{attribute 'linkalways'} 
{attribute 'no_explicit_call' := 'This FB is a CLASS and must be accessed using methods or properties'}
{attribute 'enable_dynamic_creation'}
FUNCTION_BLOCK ChunkedRequestsManager IMPLEMENTS I_ChunkedRequestsManager
VAR
	maximumChunkSizeInBytes : UDINT;
	sessionStorage : I_SessionStorage;
	headerAccessor : I_ChunkedRequestsHeaderAccessor;
END_VAR

METHOD PRIVATE CreateChunkedRequestData : I_ChunkedRequestData
VAR_INPUT
	RequestChunkSizeInBytes : UDINT;
	RequestChunkCount : UDINT;
END_VAR
VAR
	pChunkedRequestData : POINTER TO ChunkedRequestData;
END_VAR
pChunkedRequestData := __NEW(ChunkedRequestData(ChunkSizeInBytes := RequestChunkSizeInBytes, ChunkCount := RequestChunkCount));
CreateChunkedRequestData := pChunkedRequestData^;
END_METHOD

METHOD FB_init : BOOL
VAR_INPUT
	bInitRetains : BOOL; // if TRUE, the retain variables are initialized (warm start / cold start)
	bInCopyCode : BOOL;  // if TRUE, the instance afterwards gets moved into the copy code (online change)
	MaximumChunkSizeInBytes : UDINT;
	SessionStorage : I_SessionStorage;
	HeaderAccessor : I_ChunkedRequestsHeaderAccessor;
END_VAR
THIS^.maximumChunkSizeInBytes := MaximumChunkSizeInBytes;
THIS^.sessionStorage := SessionStorage;
THIS^.headerAccessor := HeaderAccessor;
END_METHOD

METHOD PUBLIC TryHandleIncomingRequest : BOOL
VAR_INPUT
	Request : I_Request;
	Response : I_ServerResponse;
	NextMidleware : I_Middleware;
END_VAR
VAR 
	hasChunkSequenceHeader : BOOL;
	chunkSequence : DINT;
	hasChunkTotalHeader : BOOL;
	chunkTotal : DINT;
	hasMoreChunksHeader : BOOL;
	hasMoreChunks : BOOL;
	requestId : T_MAXSTRING;
	sessionId : T_MAXSTRING;
	sessionData : I_SessionData;
	chunkedRequestData : I_ChunkedRequestData;
	chunkedRequest : ChunkedRequest(Request, chunkedRequestData);
END_VAR
hasChunkSequenceHeader := headerAccessor.TryGetChunkSequenceFromRequest(Request, chunkSequence);
hasChunkTotalHeader := headerAccessor.TryGetChunkTotalFromRequest(Request, chunkTotal);
hasMoreChunksHeader := headerAccessor.TryGetHasMoreChunksFromRequest(Request, hasMoreChunks);

IF (NOT hasChunkSequenceHeader) AND (NOT hasChunkTotalHeader) AND (NOT hasMoreChunksHeader) THEN
	// this is not a chunked request, simply return and it will be handled by the next middleware automatically.
	RETURN;
END_IF

// when reaching here we know that the request has at least one of the headers associated with chunked requests
// from this point on, we simply validate until we know we have all the required parts. 

IF NOT hasChunkSequenceHeader THEN
	response.Error('INVALID_CHUNK_HEADER','Chunked Request found, but chunk sequence header data is missing');
	TryHandleIncomingRequest := TRUE;
	RETURN;
END_IF

IF chunkSequence = 0 THEN
	response.Error('INVALID_CHUNK_HEADER','Chunk sequence 0 received, chunks must start from 1');
	TryHandleIncomingRequest := TRUE;
	RETURN;
END_IF

IF NOT hasChunkTotalHeader THEN
	response.Error('INVALID_CHUNK_HEADER','Chunked Request found, but chunk total header data is missing');
	TryHandleIncomingRequest := TRUE;
	RETURN;
END_IF

IF chunkSequence > chunkTotal THEN
	response.Error('INVALID_CHUNK_HEADER','Chunk sequence is greater than the chunk total');
	TryHandleIncomingRequest := TRUE;
	RETURN;
END_IF

IF NOT hasMoreChunksHeader THEN
	response.Error('INVALID_CHUNK_HEADER','Chunked Request found, but has more chunks header data is missing');
	TryHandleIncomingRequest := TRUE;
	RETURN;
END_IF

IF NOT headerAccessor.TryGetRequestIdFromRequest(Request, requestId) THEN
	response.Error('INVALID_CHUNK_HEADER','Chunked Request found, but request id header data is missing');
	TryHandleIncomingRequest := TRUE;
	RETURN;
END_IF

IF NOT headerAccessor.TryGetSessionIdFromRequest(Request, sessionId) THEN
	response.Error('INVALID_CHUNK_HEADER','Chunked Request found, but session id header data is missing');
	TryHandleIncomingRequest := TRUE;
	RETURN;
END_IF

// at this point we know we have all of the data required for handling a chunked request

IF NOT sessionStorage.TryRetrieveSessionDataById(sessionId, requestId, sessionData) THEN	
	chunkedRequestData := CreateChunkedRequestData(maximumChunkSizeInBytes, DINT_TO_UDINT(chunkTotal));
	sessionStorage.TryStoreSessionDataById(sessionId, requestId, chunkedRequestData);
ELSIF NOT __QUERYINTERFACE(sessionData, chunkedRequestData) THEN
	response.Error('SERVER_INTERNAL_ERROR','Server was unable to retreive previous session data as chunked request data');
	TryHandleIncomingRequest := TRUE;
	RETURN;
END_IF

IF NOT chunkedRequestData.TryAddChunkedPayload(request.PayloadAddress, request.PayloadSizeInBytes, chunkSequence) THEN
	response.Error('SERVER_INTERNAL_ERROR','Unable to store request payload in chunk session storage');
	sessionStorage.DisposeSessionDataById(sessionId, requestId);
	TryHandleIncomingRequest := TRUE;
	RETURN;
END_IF

IF NOT chunkedRequestData.IsComplete THEN
	Response.Accepted();
	TryHandleIncomingRequest := TRUE;
	RETURN;
END_IF

NextMidleware.Handle(chunkedRequest, Response);
sessionStorage.DisposeSessionDataById(sessionId, requestId);
TryHandleIncomingRequest := TRUE;
END_METHOD

END_FUNCTION_BLOCK

(* stored: Version 1.1.0.1, ProductVersion 3.1.4026.18
   POU ChunkedRequestsManager: Id {29bb4d2a-f5bc-4a92-b01f-999fe0b31eb2}, SpecialFunc None
   Folder Constructor: Id {2a6d5a50-12c4-4970-9247-9adefe70ce3a}
   Folder Private: Id {b0545a68-e56f-4515-abb2-33725a0e12ec}
   Method CreateChunkedRequestData: Id {3244243b-cd80-445c-b49f-744998fc8f3e}
   Method FB_init: Id {9d221340-0f02-4827-99f4-096eb3b9ae1b}
   Method TryHandleIncomingRequest: Id {7553d6da-3fdb-4ace-9b51-542f5643233e} *)
